FUNCTION_BLOCK FB_Inverter
VAR
	rAnalogSV				AT %Q* : REAL;
	
	rAxisPV					AT %I* : REAL;
	
	bClockwise				AT %Q* : BOOL;
	bCounterClockwise		AT %Q* : BOOL;
	
END_VAR

PROPERTY Analog : REAL
SET
rAnalogSV := Analog;
END_SET
END_PROPERTY

PROPERTY Axis : REAL
GET
Axis := rAxisPV;
END_GET
END_PROPERTY

PROPERTY Clockwise : BOOL
SET
bClockwise := Clockwise;
END_SET
END_PROPERTY

PROPERTY CounterClockwise : BOOL
SET
bCounterClockwise := CounterClockwise;
END_SET
END_PROPERTY

END_FUNCTION_BLOCK

(* stored: Version 1.1.0.1, ProductVersion 3.1.4024.12
   POU FB_Inverter: Id {37e3d66b-57d4-4179-a392-a5c4f3d33ef4}, SpecialFunc None
   Folder Properties: Id {1ffefa29-5b6e-4fc5-8118-b43e9a331404}
   Property Analog: Id {05c77672-fafb-457b-8eaf-1b3adc177bf0}
   Set Set: Id {2bba6512-491b-4b3a-85b5-4ab6a5a68d62}
   Property Axis: Id {74ff5bf7-a994-484d-8cd3-86a2cf109568}
   Get Get: Id {48e15fdf-c762-4035-85bf-551b24084ba3}
   Property Clockwise: Id {74f5a62b-e48d-4e1f-ac8f-224de374f152}
   Set Set: Id {6c39081f-0bc3-4a56-831a-ab8752cc3397}
   Property CounterClockwise: Id {e177ea8f-fb6e-495f-95bc-a19714d4ff59}
   Set Set: Id {661ce01c-de9f-4257-968b-3a7899fa3ffd} *)
